INTERFACE I_MotionDrive

METHOD ClearVars
VAR_INPUT
    Done : BOOL;
END_VAR
END_METHOD

PROPERTY EnableMode : ENUM_StageEnableMode
GET
END_GET
SET
END_SET
END_PROPERTY

PROPERTY Name : STRING
GET
END_GET
SET
END_SET
END_PROPERTY

METHOD PreMoveHandling
VAR_INPUT
END_VAR
END_METHOD

METHOD RestoreSettings
VAR_INPUT
END_VAR
END_METHOD

METHOD  UpdateParamAndStatus
VAR_INPUT
END_VAR
END_METHOD

END_INTERFACE

(* stored: Version 1.1.0.1
   Itf I_MotionDrive: Id {848572bc-fef8-4708-bb80-0dc37710e2cf}
   Method ClearVars: Id {4b5fb135-307e-42cf-967b-f614dbd2b225}
   Property EnableMode: Id {adfca8af-3f45-4930-b0c2-1c641071c27e}
   Get Get: Id {cb007901-22fb-4dd1-a7e8-913e722e45c4}
   Set Set: Id {f302ffc4-bf3a-4fcc-9730-7c3f1c68c572}
   Property Name: Id {d0be49c7-7763-48e4-931a-0ecf586b19f0}
   Get Get: Id {dfedf110-1b25-46e5-a039-730cf49e342e}
   Set Set: Id {e91d6d3d-7a85-4e7f-8abb-cb3d9c8eac57}
   Method PreMoveHandling: Id {9d2919b9-444e-4c31-9bbe-e53274fd277d}
   Method RestoreSettings: Id {14eecb93-a536-495b-8a81-ca4fbc68ea55}
   Method UpdateParamAndStatus: Id {e7e24ac1-a3db-410d-b1d8-9f1d070d6f33} *)
